FUNCTION_BLOCK _ULINT_TestSuite EXTENDS TcUnit.FB_TestSuite
VAR
END_VAR

TestAddress();
TestClearReference();
TestClone();
TestTypeNameReturnsExpected();
TestIsFloat();
TestIsSigned();
TestMakeReferenceToFollowsReference();
TestMakeReferenceToUpdatesReference();
TestSize();
TestValueReturnsExpectedAfterInit();
TestValueReturnsExpectedAfterChange();
TestSerializeTypeWith();
TestSerializeWith();
TestTryDeserializeFrom();
TestTryMakeReferenceToFollowsReference();
TestTryMakeReferenceToUpdatesReference();

METHOD PUBLIC TestAddress
VAR
    _type : _ULINT(0);
    notExpected : PVOID := 0;
    actual : PVOID;
END_VAR
TEST('TestAddress');

actual := _type.Address;

AssertFalse(
    Condition := (notExpected = actual),
    Message := 'Type did not return a valid address.'
);

TEST_FINISHED();
END_METHOD

METHOD PUBLIC TestClearReference
VAR
    _type : _ULINT(0);
	target : ULINT := 0;
    expected : ULINT := 0;
    actual : ULINT;
END_VAR
TEST('TestClearReference');

_type.MakeReferenceTo(target);
_type.ClearReference();
target := 123;

actual := _type.Value;

AssertEquals(
    Expected := expected,
    Actual := actual,
    Message := 'Value did not follow target change'
);

TEST_FINISHED();
END_METHOD

METHOD PUBLIC TestClone
VAR
    _type : _ULINT(123);
	clone : I_Datatype;
	isValidClone : BOOL;
	compareResult : DINT;
END_VAR
TEST('TestClone');

clone := _type.Clone();

isValidClone := clone <> 0;

IF isValidClone THEN
	compareResult := memcmp(_type.Address, clone.Address, clone.Size);
END_IF

AssertTrue(
	Condition := isValidClone,
	Message := 'Clone did not produce a clone'
);

AssertEquals_DINT(
	Expected := 0,
    Actual := compareResult,
    Message := 'Clone did not return a valid clone.'
);

clone.Dispose();

TEST_FINISHED();
END_METHOD

METHOD PUBLIC TestIsFloat
VAR
    _type : _ULINT(0);
END_VAR
TEST('TestIsFloat');

AssertFalse(
	Condition := _type.IsFloat,
    Message := 'Type did not correctly identify itself as being unsigned'
);

TEST_FINISHED();
END_METHOD

METHOD PUBLIC TestIsSigned
VAR
    _type : _ULINT(0);
END_VAR
TEST('TestIsSigned');

AssertFalse(
	Condition := _type.IsSigned,
    Message := 'Type did not correctly identify itself as being unsigned'
);

TEST_FINISHED();
END_METHOD

METHOD PUBLIC TestMakeReferenceToFollowsReference
VAR
    _type : _ULINT(0);
	target : ULINT := 0;
    expected : ULINT := 123;
    actual : ULINT;
END_VAR
TEST('TestMakeReferenceToFollowsReference');

_type.MakeReferenceTo(target);
target := 123;

actual := _type.Value;

AssertEquals(
    Expected := expected,
    Actual := actual,
    Message := 'Value did not follow target change'
);

TEST_FINISHED();
END_METHOD

METHOD PUBLIC TestMakeReferenceToUpdatesReference
VAR
    _type : _ULINT(0);
	target : ULINT := 0;
    expected : ULINT := 123;
    actual : ULINT;
END_VAR
TEST('TestMakeReferenceToUpdatesReference');

_type.MakeReferenceTo(target);
_type.Value := 123;

actual := target;

AssertEquals(
    Expected := expected,
    Actual := actual,
    Message := 'Value did not update target'
);

TEST_FINISHED();
END_METHOD

METHOD PUBLIC TestSerializeTypeWith
VAR
    _type : _ULINT(0);
    serializer : JsonSerializer;
    expected : STRING(500) := '{"typeName":"ULINT","minValue":0,"maxValue":18446744073709551615,"isSigned":false,"isFloat":false}';
    actual : STRING(500);
END_VAR
TEST('TestSerializeTypeWith');

serializer.Reset();
_type.SerializeTypeWith(serializer);
serializer.TryGetSerializedData(ADR(actual), SIZEOF(actual));

AssertEquals_STRING(
    Expected := expected,
    Actual := actual,
    Message := 'Serialization of type did not return correct string.'
);

TEST_FINISHED();
END_METHOD

METHOD PUBLIC TestSerializeWith
VAR
    _type : _ULINT(32767);
    serializer : JsonSerializer;
    expected : STRING := '32767';
    actual : STRING(500);
END_VAR
TEST('TestSerializeWith');

serializer.Reset();
_type.SerializeWith(serializer);
serializer.TryGetSerializedData(ADR(actual), SIZEOF(actual));

AssertEquals_STRING(
    Expected := expected,
    Actual := actual,
    Message := 'Serialization of type data did not return correct string.'
);

TEST_FINISHED();
END_METHOD

METHOD PUBLIC TestSize
VAR
    _type : _ULINT(0);
    expected : UDINT := SIZEOF(ULINT);
    actual : UDINT;
END_VAR
TEST('TestSize');

actual := _type.Size;

AssertEquals_UDINT(
    Expected := Expected,
    Actual := actual,
    Message := 'Type did not return the correct size.'
);

TEST_FINISHED();
END_METHOD

METHOD PUBLIC TestTryDeserializeFrom
VAR
    deserializer : JsonDeserializer;
    feedback : DeserializerFeedback;
    json : STRING := '32767';
    _type : _ULINT(0);
    expected : ULINT := 32767;
    actual : ULINT;
 END_VAR
TEST('TestTryDeserializeFrom');

deserializer.Reset();
deserializer.TryLoad(json);
_type.TryDeserializeFrom(Deserializer, Feedback);

actual := _type.Value;

AssertEquals(
    Expected := expected,
    Actual := actual,
    Message := 'Type did not deserialize correctly.'
);

TEST_FINISHED();
END_METHOD

METHOD PUBLIC TestTryMakeReferenceToFollowsReference
VAR
    _type : _ULINT(0);
	target : _ULINT(0);
    expected : ULINT := 123;
    actual : ULINT;
END_VAR
TEST('TestTryMakeReferenceToFollowsReference');

_type.TryMakeReferenceTo(target);
target.Value := 123;

actual := _type.Value;

AssertEquals(
    Expected := expected,
    Actual := actual,
    Message := 'Value did not follow target change'
);

TEST_FINISHED();
END_METHOD

METHOD PUBLIC TestTryMakeReferenceToUpdatesReference
VAR
    _type : _ULINT(0);
	target : _ULINT(0);
    expected : ULINT := 123;
    actual : ULINT;
END_VAR
TEST('TestTryMakeReferenceToUpdatesReference');

_type.TryMakeReferenceTo(target);
_type.Value := 123;

actual := target.Value;

AssertEquals(
    Expected := expected,
    Actual := actual,
    Message := 'Value did not update target'
);

TEST_FINISHED();
END_METHOD

METHOD PUBLIC TestTypeNameReturnsExpected
VAR
    _type : _ULINT(0);
    expected : STRING := 'ULINT';
    actual : STRING;
END_VAR
TEST('TestTypeNameReturnsExpected');

actual := _type.TypeName;

AssertEquals_STRING(
    Expected := expected,
    Actual := actual,
    Message := 'Type did not return correct iec type.'
);

TEST_FINISHED();
END_METHOD

METHOD PUBLIC TestValueReturnsExpectedAfterChange
VAR
    _type : _ULINT(0);
    expected : ULINT := 32767;
    actual : ULINT;
END_VAR
TEST('TestValueReturnsExpectedAfterChange');

_type.Value := 32767;

actual := _type.Value;

AssertEquals(
    Expected := expected,
    Actual := actual,
    Message := 'Expected value not returned after change.'
);

TEST_FINISHED();
END_METHOD

METHOD PUBLIC TestValueReturnsExpectedAfterInit
VAR
    _type : _ULINT(32767);
    expected : ULINT := 32767;
    actual : ULINT;
END_VAR
TEST('TestValueReturnsExpectedAfterInit');

actual := _type.Value;

AssertEquals(
    Expected := expected,
    Actual := actual,
    Message := 'Expected value not returned after Init.'
);

TEST_FINISHED();
END_METHOD

END_FUNCTION_BLOCK

(* stored: Version 1.1.0.1, ProductVersion 3.1.4024.12
   POU _ULINT_TestSuite: Id {b192cb24-11b9-4292-9714-55e8e6f12159}, SpecialFunc None
   Method TestAddress: Id {4e1ddd1e-b892-4279-b9ef-bd5a74a427a3}
   Method TestClearReference: Id {fb3a5cc9-727b-41fc-a071-b02c4e85404c}
   Method TestClone: Id {09251629-e227-41ce-bef8-149af2ac9cb2}
   Method TestIsFloat: Id {087d8886-8991-0757-0864-520aa8779b79}
   Method TestIsSigned: Id {ddfb716c-293b-4e12-941a-918eb74ffb3e}
   Method TestMakeReferenceToFollowsReference: Id {a26708d3-b980-4556-9d7b-00a4afc3d949}
   Method TestMakeReferenceToUpdatesReference: Id {642c4d0d-c4f9-48e7-a1b5-c2d6d9315062}
   Method TestSerializeTypeWith: Id {63b66417-0989-42cc-90e8-4f484b915534}
   Method TestSerializeWith: Id {9583e333-3cf6-4998-967a-2d7e456b6e29}
   Method TestSize: Id {1ed1b42a-f01d-4682-89dd-08a4d8559382}
   Method TestTryDeserializeFrom: Id {b4976324-da39-4041-895a-c9a098d5f720}
   Method TestTryMakeReferenceToFollowsReference: Id {afec9969-bf23-4003-a26c-1459f053acff}
   Method TestTryMakeReferenceToUpdatesReference: Id {72feed62-b544-420d-98a9-7258877e240e}
   Method TestTypeNameReturnsExpected: Id {d2ff9522-698e-4f4a-83ac-def1304b6608}
   Method TestValueReturnsExpectedAfterChange: Id {a568b62d-721c-4984-ae93-dc6410289335}
   Method TestValueReturnsExpectedAfterInit: Id {11d6f356-794c-4cf3-a10b-5d3d5ed91242} *)
